TYPE ST_DALIMemoryBank :
STRUCT
	sOffset			:	STRING(20);
	sName			:	STRING(255);
	nValueDec		:	BYTE;
	nValueHex		:	STRING(20);
END_STRUCT
END_TYPE

(* stored: Version 1.1.0.1, ProductVersion 3.1.4024.12
   DUT ST_DALIMemoryBank: Id {57babaf8-e52d-4b65-b291-6554c1922237} *)
